FUNCTION_BLOCK FB_TorqueSensor
VAR_INPUT
END_VAR
VAR_OUTPUT
END_VAR
VAR
END_VAR

END_FUNCTION_BLOCK

(* stored: Version 1.1.0.1, ProductVersion 3.1.4024.12
   POU FB_TorqueSensor: Id {09bd596b-a83b-46b1-b921-9eab5b868d1b}, SpecialFunc None *)
